# EPICS StreamDevice protocol: protocols/ai.proto
Terminator = LF;
ExtraInput = Ignore;

isTriggered {
	out "is_triggered";
	in "%d";
}

setEsEnable {
	out "es_enable %d";
	in;
}

getEsEnable {
	out "es_enable";
	in "%d";
}
